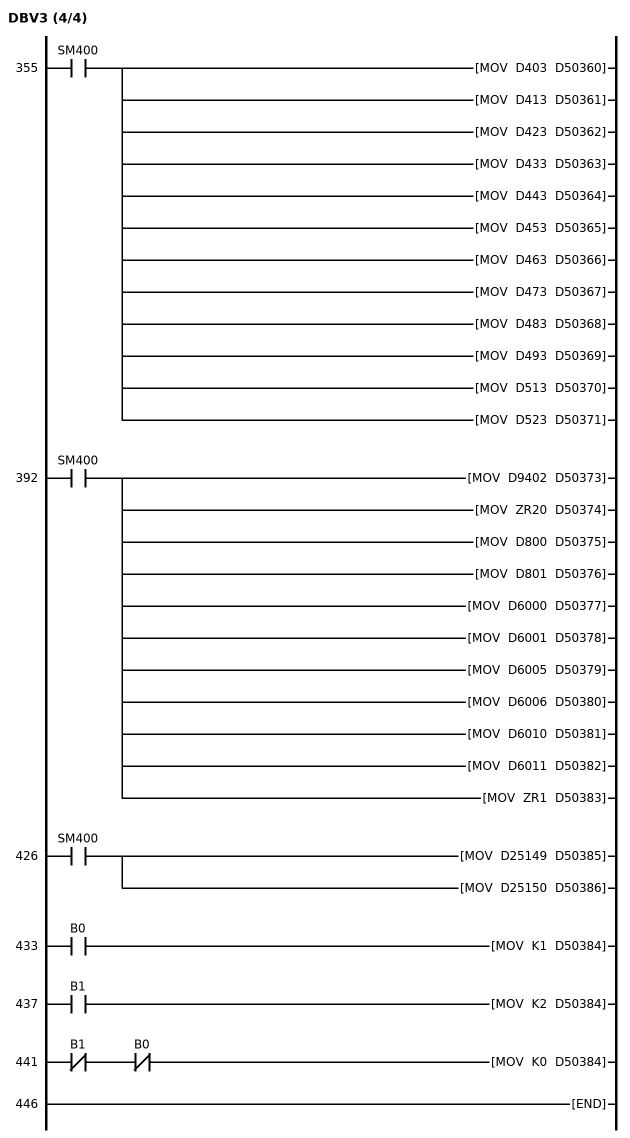
[picture p168: ladder of DBV3, rungs at steps 355 to 446]
355   LD      SM400
      MOV     D403 D50360
      MOV     D413 D50361
      MOV     D423 D50362
      MOV     D433 D50363
      MOV     D443 D50364
      MOV     D453 D50365
      MOV     D463 D50366
      MOV     D473 D50367
      MOV     D483 D50368
      MOV     D493 D50369
      MOV     D513 D50370
      MOV     D523 D50371
392   LD      SM400
      MOV     D9402 D50373
      MOV     ZR20 D50374
      MOV     D800 D50375
      MOV     D801 D50376
      MOV     D6000 D50377
      MOV     D6001 D50378
      MOV     D6005 D50379
      MOV     D6006 D50380
      MOV     D6010 D50381
      MOV     D6011 D50382
      MOV     ZR1 D50383
426   LD      SM400
      MOV     D25149 D50385
      MOV     D25150 D50386
433   LD      B0
      MOV     K1 D50384
437   LD      B1
      MOV     K2 D50384
441   LDI     B1
      ANI     B0
      MOV     K0 D50384
446   END
END_PROGRAM

PROGRAM dryer_cover
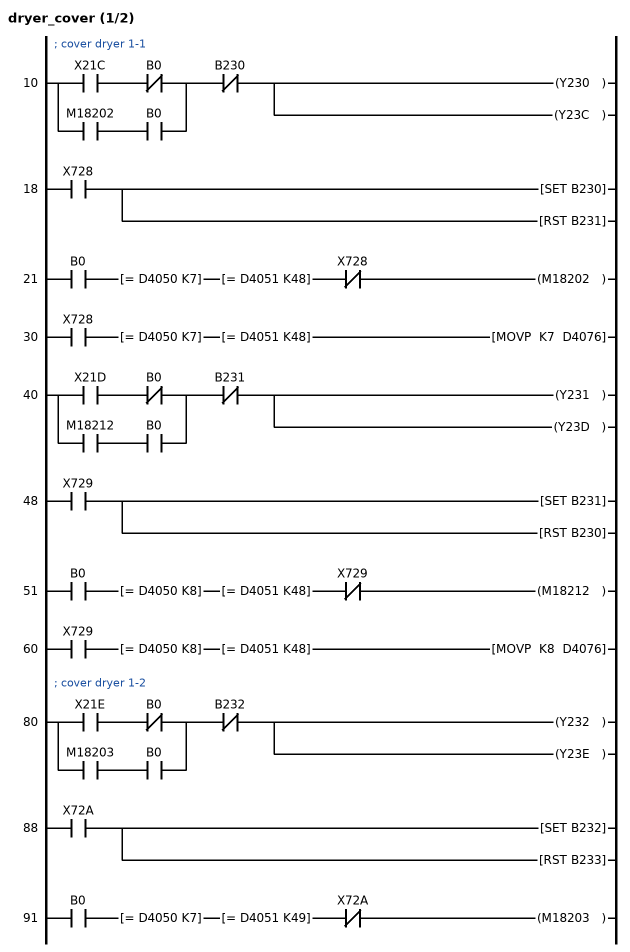
; cover dryer 1-1
10    LD      X21C
      ANI     B0
      LD      M18202
      AND     B0
      ORB
      ANI     B230
      OUT     Y230
      OUT     Y23C
18    LD      X728
      SET     B230
      RST     B231
21    LD      B0
      AND=    D4050 K7
      AND=    D4051 K48
      ANI     X728
      OUT     M18202
30    LD      X728
      AND=    D4050 K7
      AND=    D4051 K48
      MOVP    K7 D4076
40    LD      X21D
      ANI     B0
      LD      M18212
      AND     B0
      ORB
      ANI     B231
      OUT     Y231
      OUT     Y23D
48    LD      X729
      SET     B231
      RST     B230
51    LD      B0
      AND=    D4050 K8
      AND=    D4051 K48
      ANI     X729
      OUT     M18212
60    LD      X729
      AND=    D4050 K8
      AND=    D4051 K48
      MOVP    K8 D4076
; cover dryer 1-2
80    LD      X21E
      ANI     B0
      LD      M18203
      AND     B0
      ORB
      ANI     B232
      OUT     Y232
      OUT     Y23E
88    LD      X72A
      SET     B232
      RST     B233
91    LD      B0
      AND=    D4050 K7
      AND=    D4051 K49
      ANI     X72A
      OUT     M18203
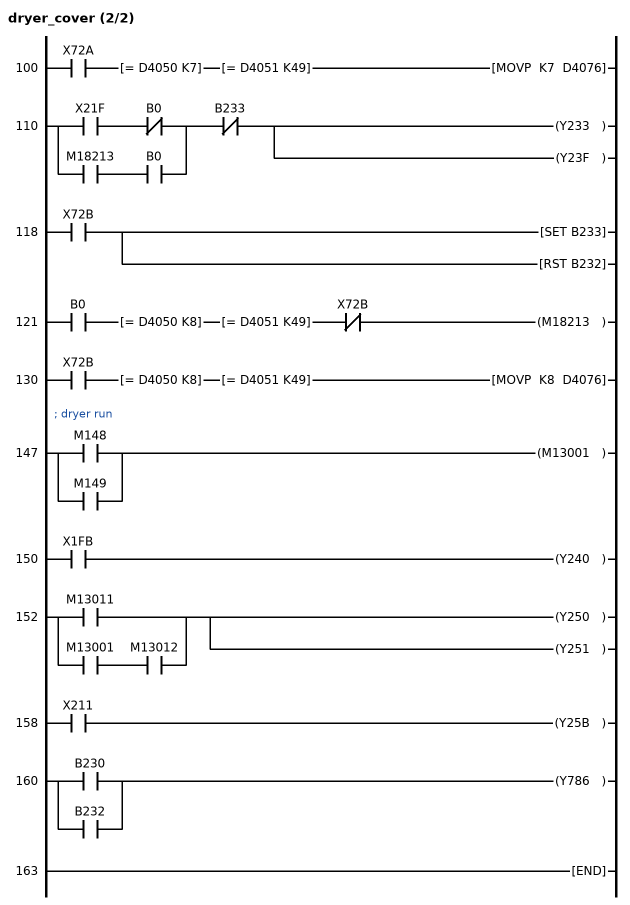
100   LD      X72A
      AND=    D4050 K7
      AND=    D4051 K49
      MOVP    K7 D4076
110   LD      X21F
      ANI     B0
      LD      M18213
      AND     B0
      ORB
      ANI     B233
      OUT     Y233
      OUT     Y23F
118   LD      X72B
      SET     B233
      RST     B232
121   LD      B0
      AND=    D4050 K8
      AND=    D4051 K49
      ANI     X72B
      OUT     M18213
130   LD      X72B
      AND=    D4050 K8
      AND=    D4051 K49
      MOVP    K8 D4076
; dryer run
147   LD      M148
      OR      M149
      OUT     M13001
150   LD      X1FB
      OUT     Y240
152   LD      M13011
      LD      M13001
      AND     M13012
      ORB
      OUT     Y250
      OUT     Y251
158   LD      X211
      OUT     Y25B
160   LD      B230
      OR      B232
      OUT     Y786
163   END
END_PROGRAM

FUNCTION_BLOCK I+ST_4f96081e274e4d1c
VAR_INPUT
  __IST_EN_IN : BOOL;
END_VAR
VAR_OUTPUT
  __IST_EN_OUT : BOOL;
END_VAR
(* IST HEADER START *)
IF NOT __IST_EN_IN THEN __IST_EN_OUT:=FALSE; RETURN; END_IF;
(* VERSION=1:TYPE=STB *)
(* IST HEADER END *)
D3016 := D3006 / k10 ;
END_FUNCTION_BLOCK

FUNCTION_BLOCK I+ST_76367eaf8b844e8d
VAR_INPUT
  __IST_EN_IN : BOOL;
END_VAR
VAR_OUTPUT
  __IST_EN_OUT : BOOL;
END_VAR
(* IST HEADER START *)
IF NOT __IST_EN_IN THEN __IST_EN_OUT:=FALSE; RETURN; END_IF;
(* VERSION=1:TYPE=STB *)
(* IST HEADER END *)
D3015 := D3006 / k10 ;
END_FUNCTION_BLOCK

FUNCTION_BLOCK I+ST_b7c0c6d72a974ae8
VAR_INPUT
  __IST_EN_IN : BOOL;
END_VAR
VAR_OUTPUT
  __IST_EN_OUT : BOOL;
END_VAR
(* IST HEADER START *)
IF NOT __IST_EN_IN THEN __IST_EN_OUT:=FALSE; RETURN; END_IF;
(* VERSION=1:TYPE=STB *)
(* IST HEADER END *)
ZR1010000Z9 := k0 ;
ZR1020000Z9:= k0 ;
ZR1030000Z9 := k0 ;
ZR1040000Z9 := k0 ;
ZR1050000Z9 := k0 ;
ZR1060000Z9 := k0 ;
ZR1070000Z9 := k0 ;
ZR1080000Z9 := k0 ;
ZR1090000Z9 := k0 ;
ZR1100000Z9 := k0 ;
ZR1110000Z9 := k0 ;
ZR1120000Z9 := k0 ;
ZR1130000Z9 := k0 ;
ZR1140000Z9 := k0 ;
ZR1150000Z9 := k0 ;
ZR1160000Z9 := k0 ;
ZR1170000Z9 := k0 ;
ZR1180000Z9 := k0 ;
ZR1190000Z9 := k0 ;
ZR1200000Z9 := k0 ;
ZR1210000Z9 := k0 ;
ZR1220000Z9 := k0 ;
ZR1230000Z9 := k0 ;
ZR1240000Z9 := k0 ;
ZR1250000Z9 := k0 ;
ZR1260000Z9 := k0 ;
ZR1270000Z9 := k0 ;
ZR1280000Z9 := k0 ;
ZR1290000Z9 := k0 ;
ZR1300000Z9 := k0 ;
ZR1310000Z9 := k0 ;
ZR1320000Z9 := k0 ;
ZR1330000Z9 := k0 ;
ZR1340000Z9 := k0 ;
ZR1350000Z9 := k0 ;
ZR1360000Z9 := k0 ;
ZR1370000Z9 := k0 ;
ZR1380000Z9 := k0 ;
ZR1390000Z9 := k0 ;
ZR1400000Z9 := k0 ;
ZR1410000Z9 := k0 ;
ZR1420000Z9 := k0 ;
ZR1430000Z9 := k0 ;
ZR1440000Z9 := k0 ;
ZR1450000Z9 := k0 ;
ZR1460000Z9 := k0 ;
ZR1470000Z9 := k0 ;
ZR1480000Z9 := k0 ;
ZR1490000Z9 := k0 ;
ZR1500000Z9 := k0 ;
ZR1510000Z9 := k0 ;
ZR1520000Z9 := k0 ;
ZR1530000Z9 := k0 ;
ZR1540000Z9 := k0 ;
ZR1550000Z9 := k0 ;
ZR1560000Z9 := k0 ;
ZR1570000Z9 := k0 ;
ZR1580000Z9 := k0 ;
ZR1590000Z9 := k0 ;
ZR1600000Z9 := k0 ;
END_FUNCTION_BLOCK

FUNCTION_BLOCK I+ST_f649ea45d16546a8
VAR_INPUT
  __IST_EN_IN : BOOL;
END_VAR
VAR_OUTPUT
  __IST_EN_OUT : BOOL;
END_VAR
(* IST HEADER START *)
IF NOT __IST_EN_IN THEN __IST_EN_OUT:=FALSE; RETURN; END_IF;
(* VERSION=1:TYPE=STB *)
(* IST HEADER END *)
ZR1610000Z9 := k0 ;
ZR1620000Z9 := k0 ;
ZR1630000Z9 := k0 ;
ZR1640000Z9 := k0 ;
ZR1650000Z9 := k0 ;
ZR1660000Z9 := k0 ;
ZR1670000Z9 := k0 ;
ZR1680000Z9 := k0 ;
ZR1690000Z9 := k0 ;

ZR1800000Z9 := k0 ;
ZR1810000Z9 := k0 ;
ZR1820000Z9 := k0 ;
ZR1830000Z9 := k0 ;
ZR1840000Z9 := k0 ;
ZR1850000Z9 := k0 ;
ZR1860000Z9 := k0 ;
ZR1870000Z9 := k0 ;
ZR1880000Z9 := k0 ;
ZR1890000Z9 := k0 ;
ZR1900000Z9 := k0 ;
END_FUNCTION_BLOCK

PROGRAM POU_01
0     END
END_PROGRAM

PROGRAM pro_time
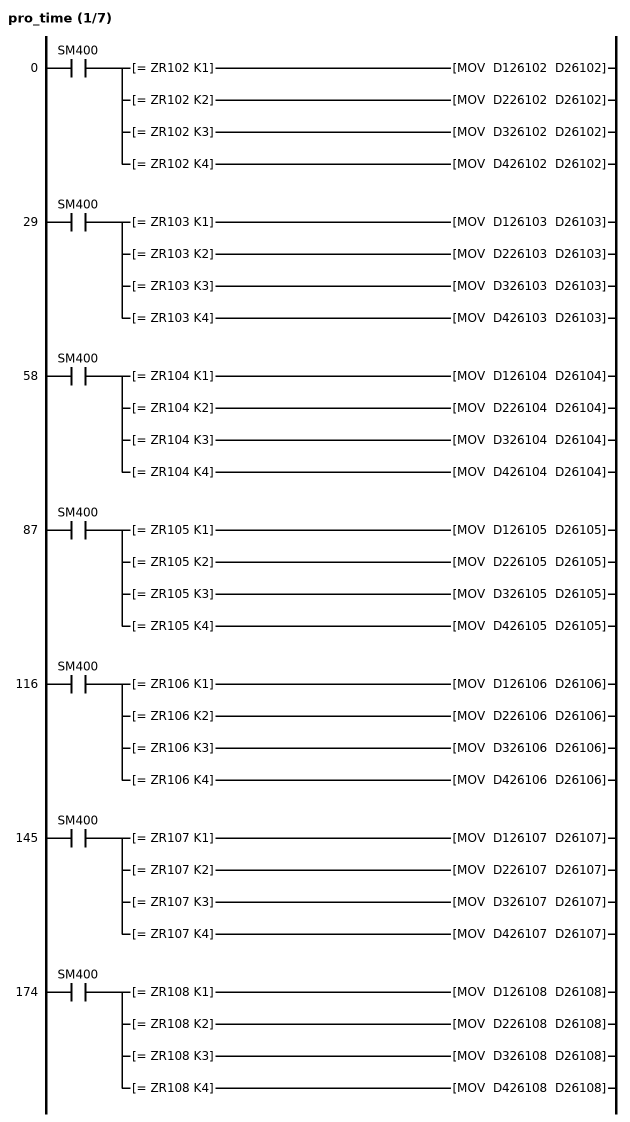
0     LD      SM400
      MPS
      AND=    ZR102 K1
      MOV     D126102 D26102
      MRD
      AND=    ZR102 K2
      MOV     D226102 D26102
      MRD
      AND=    ZR102 K3
      MOV     D326102 D26102
      MPP
      AND=    ZR102 K4
      MOV     D426102 D26102
29    LD      SM400
      MPS
      AND=    ZR103 K1
      MOV     D126103 D26103
      MRD
      AND=    ZR103 K2
      MOV     D226103 D26103
      MRD
      AND=    ZR103 K3
      MOV     D326103 D26103
      MPP
      AND=    ZR103 K4
      MOV     D426103 D26103
58    LD      SM400
      MPS
      AND=    ZR104 K1
      MOV     D126104 D26104
      MRD
      AND=    ZR104 K2
      MOV     D226104 D26104
      MRD
      AND=    ZR104 K3
      MOV     D326104 D26104
      MPP
      AND=    ZR104 K4
      MOV     D426104 D26104
87    LD      SM400
      MPS
      AND=    ZR105 K1
      MOV     D126105 D26105
      MRD
      AND=    ZR105 K2
      MOV     D226105 D26105
      MRD
      AND=    ZR105 K3
      MOV     D326105 D26105
      MPP
      AND=    ZR105 K4
      MOV     D426105 D26105
116   LD      SM400
      MPS
      AND=    ZR106 K1
      MOV     D126106 D26106
      MRD
      AND=    ZR106 K2
      MOV     D226106 D26106
      MRD
      AND=    ZR106 K3
      MOV     D326106 D26106
      MPP
      AND=    ZR106 K4
      MOV     D426106 D26106
145   LD      SM400
      MPS
      AND=    ZR107 K1
      MOV     D126107 D26107
      MRD
      AND=    ZR107 K2
      MOV     D226107 D26107
      MRD
      AND=    ZR107 K3
      MOV     D326107 D26107
      MPP
      AND=    ZR107 K4
      MOV     D426107 D26107
174   LD      SM400
      MPS
      AND=    ZR108 K1
      MOV     D126108 D26108
      MRD
      AND=    ZR108 K2
      MOV     D226108 D26108
      MRD
      AND=    ZR108 K3
      MOV     D326108 D26108
      MPP
      AND=    ZR108 K4
      MOV     D426108 D26108
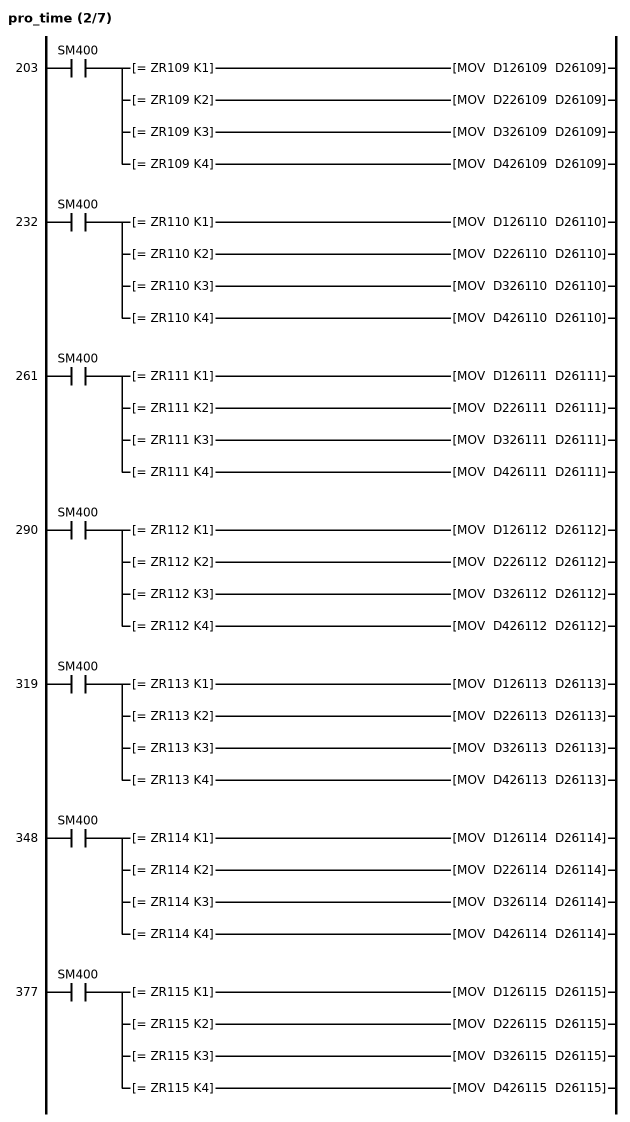
203   LD      SM400
      MPS
      AND=    ZR109 K1
      MOV     D126109 D26109
      MRD
      AND=    ZR109 K2
      MOV     D226109 D26109
      MRD
      AND=    ZR109 K3
      MOV     D326109 D26109
      MPP
      AND=    ZR109 K4
      MOV     D426109 D26109
232   LD      SM400
      MPS
      AND=    ZR110 K1
      MOV     D126110 D26110
      MRD
      AND=    ZR110 K2
      MOV     D226110 D26110
      MRD
      AND=    ZR110 K3
      MOV     D326110 D26110
      MPP
      AND=    ZR110 K4
      MOV     D426110 D26110
261   LD      SM400
      MPS
      AND=    ZR111 K1
      MOV     D126111 D26111
      MRD
      AND=    ZR111 K2
      MOV     D226111 D26111
      MRD
      AND=    ZR111 K3
      MOV     D326111 D26111
      MPP
      AND=    ZR111 K4
      MOV     D426111 D26111
290   LD      SM400
      MPS
      AND=    ZR112 K1
      MOV     D126112 D26112
      MRD
      AND=    ZR112 K2
      MOV     D226112 D26112
      MRD
      AND=    ZR112 K3
      MOV     D326112 D26112
      MPP
      AND=    ZR112 K4
      MOV     D426112 D26112
319   LD      SM400
      MPS
      AND=    ZR113 K1
      MOV     D126113 D26113
      MRD
      AND=    ZR113 K2
      MOV     D226113 D26113
      MRD
      AND=    ZR113 K3
      MOV     D326113 D26113
      MPP
      AND=    ZR113 K4
      MOV     D426113 D26113
348   LD      SM400
      MPS
      AND=    ZR114 K1
      MOV     D126114 D26114
      MRD
      AND=    ZR114 K2
      MOV     D226114 D26114
      MRD
      AND=    ZR114 K3
      MOV     D326114 D26114
      MPP
      AND=    ZR114 K4
      MOV     D426114 D26114
377   LD      SM400
      MPS
      AND=    ZR115 K1
      MOV     D126115 D26115
      MRD
      AND=    ZR115 K2
      MOV     D226115 D26115
      MRD
      AND=    ZR115 K3
      MOV     D326115 D26115
      MPP
      AND=    ZR115 K4
      MOV     D426115 D26115
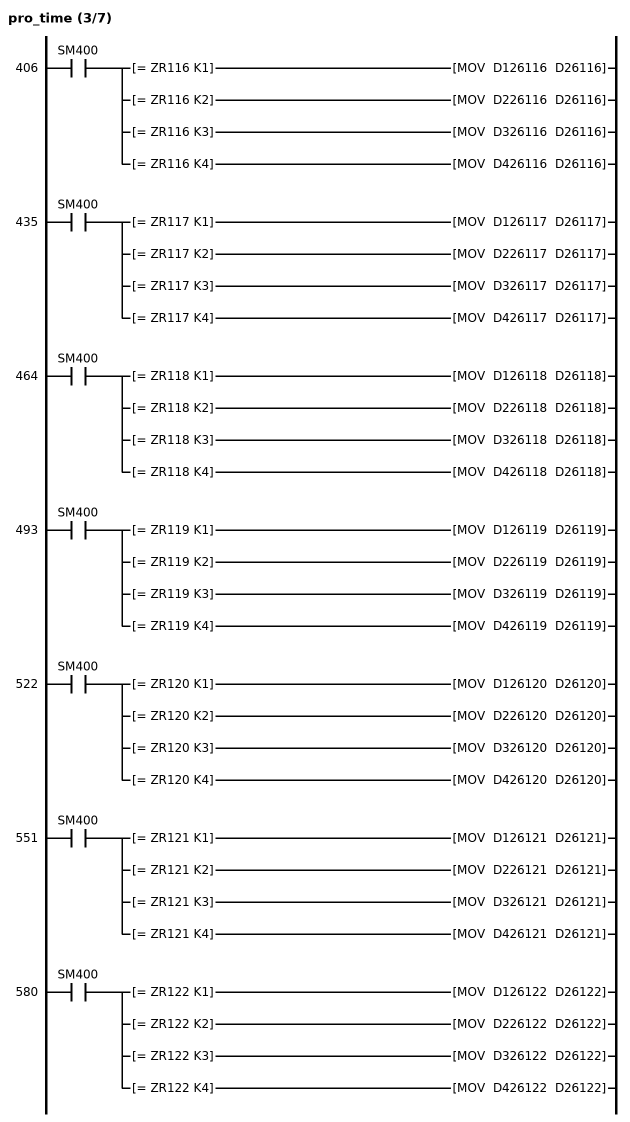
406   LD      SM400
      MPS
      AND=    ZR116 K1
      MOV     D126116 D26116
      MRD
      AND=    ZR116 K2
      MOV     D226116 D26116
      MRD
      AND=    ZR116 K3
      MOV     D326116 D26116
      MPP
      AND=    ZR116 K4
      MOV     D426116 D26116
435   LD      SM400
      MPS
      AND=    ZR117 K1
      MOV     D126117 D26117
      MRD
      AND=    ZR117 K2
      MOV     D226117 D26117
      MRD
      AND=    ZR117 K3
      MOV     D326117 D26117
      MPP
      AND=    ZR117 K4
      MOV     D426117 D26117
464   LD      SM400
      MPS
      AND=    ZR118 K1
      MOV     D126118 D26118
      MRD
      AND=    ZR118 K2
      MOV     D226118 D26118
      MRD
      AND=    ZR118 K3
      MOV     D326118 D26118
      MPP
      AND=    ZR118 K4
      MOV     D426118 D26118
493   LD      SM400
      MPS
      AND=    ZR119 K1
      MOV     D126119 D26119
      MRD
      AND=    ZR119 K2
      MOV     D226119 D26119
      MRD
      AND=    ZR119 K3
      MOV     D326119 D26119
      MPP
      AND=    ZR119 K4
      MOV     D426119 D26119
522   LD      SM400
      MPS
      AND=    ZR120 K1
      MOV     D126120 D26120
      MRD
      AND=    ZR120 K2
      MOV     D226120 D26120
      MRD
      AND=    ZR120 K3
      MOV     D326120 D26120
      MPP
      AND=    ZR120 K4
      MOV     D426120 D26120
551   LD      SM400
      MPS
      AND=    ZR121 K1
      MOV     D126121 D26121
      MRD
      AND=    ZR121 K2
      MOV     D226121 D26121
      MRD
      AND=    ZR121 K3
      MOV     D326121 D26121
      MPP
      AND=    ZR121 K4
      MOV     D426121 D26121
580   LD      SM400
      MPS
      AND=    ZR122 K1
      MOV     D126122 D26122
      MRD
      AND=    ZR122 K2
      MOV     D226122 D26122
      MRD
      AND=    ZR122 K3
      MOV     D326122 D26122
      MPP
      AND=    ZR122 K4
      MOV     D426122 D26122
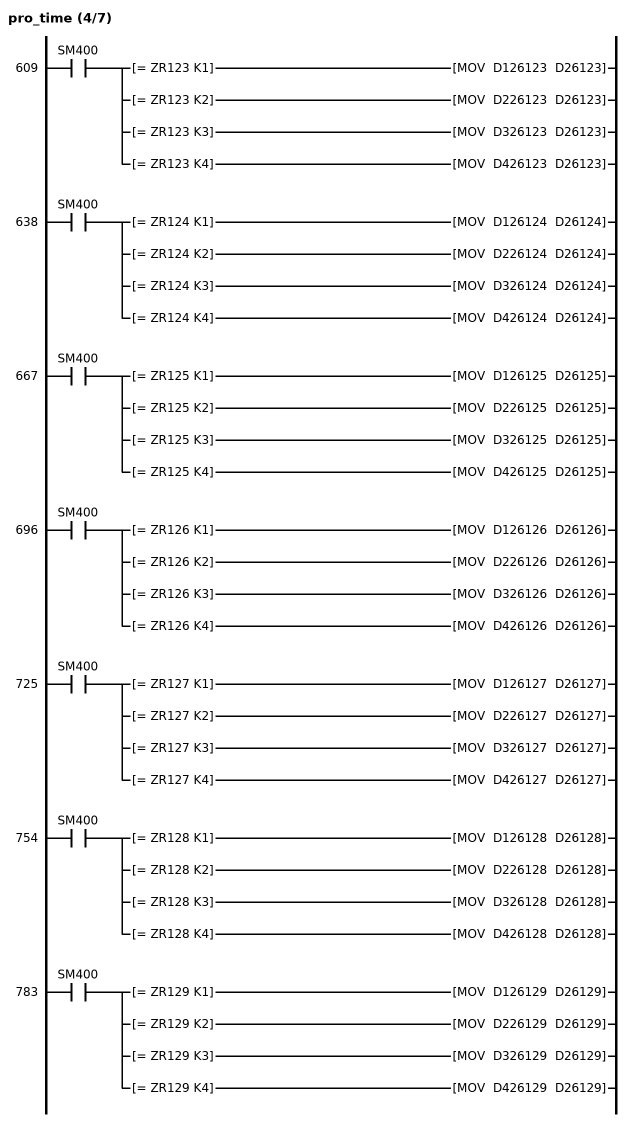
609   LD      SM400
      MPS
      AND=    ZR123 K1
      MOV     D126123 D26123
      MRD
      AND=    ZR123 K2
      MOV     D226123 D26123
      MRD
      AND=    ZR123 K3
      MOV     D326123 D26123
      MPP
      AND=    ZR123 K4
      MOV     D426123 D26123
638   LD      SM400
      MPS
      AND=    ZR124 K1
      MOV     D126124 D26124
      MRD
      AND=    ZR124 K2
      MOV     D226124 D26124
      MRD
      AND=    ZR124 K3
      MOV     D326124 D26124
      MPP
      AND=    ZR124 K4
      MOV     D426124 D26124
667   LD      SM400
      MPS
      AND=    ZR125 K1
      MOV     D126125 D26125
      MRD
      AND=    ZR125 K2
      MOV     D226125 D26125
      MRD
      AND=    ZR125 K3
      MOV     D326125 D26125
      MPP
      AND=    ZR125 K4
      MOV     D426125 D26125
696   LD      SM400
      MPS
      AND=    ZR126 K1
      MOV     D126126 D26126
      MRD
      AND=    ZR126 K2
      MOV     D226126 D26126
      MRD
      AND=    ZR126 K3
      MOV     D326126 D26126
      MPP
      AND=    ZR126 K4
      MOV     D426126 D26126
725   LD      SM400
      MPS
      AND=    ZR127 K1
      MOV     D126127 D26127
      MRD
      AND=    ZR127 K2
      MOV     D226127 D26127
      MRD
      AND=    ZR127 K3
      MOV     D326127 D26127
      MPP
      AND=    ZR127 K4
      MOV     D426127 D26127
754   LD      SM400
      MPS
      AND=    ZR128 K1
      MOV     D126128 D26128
      MRD
      AND=    ZR128 K2
      MOV     D226128 D26128
      MRD
      AND=    ZR128 K3
      MOV     D326128 D26128
      MPP
      AND=    ZR128 K4
      MOV     D426128 D26128
783   LD      SM400
      MPS
      AND=    ZR129 K1
      MOV     D126129 D26129
      MRD
      AND=    ZR129 K2
      MOV     D226129 D26129
      MRD
      AND=    ZR129 K3
      MOV     D326129 D26129
      MPP
      AND=    ZR129 K4
      MOV     D426129 D26129
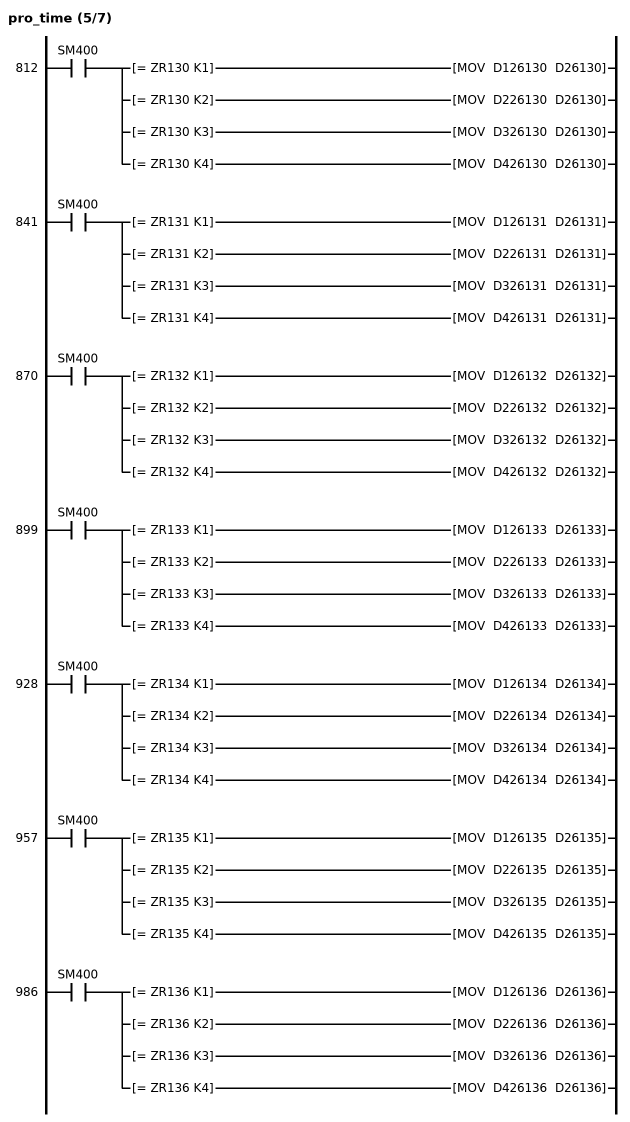
812   LD      SM400
      MPS
      AND=    ZR130 K1
      MOV     D126130 D26130
      MRD
      AND=    ZR130 K2
      MOV     D226130 D26130
      MRD
      AND=    ZR130 K3
      MOV     D326130 D26130
      MPP
      AND=    ZR130 K4
      MOV     D426130 D26130
841   LD      SM400
      MPS
      AND=    ZR131 K1
      MOV     D126131 D26131
      MRD
      AND=    ZR131 K2
      MOV     D226131 D26131
      MRD
      AND=    ZR131 K3
      MOV     D326131 D26131
      MPP
      AND=    ZR131 K4
      MOV     D426131 D26131
870   LD      SM400
      MPS
      AND=    ZR132 K1
      MOV     D126132 D26132
      MRD
      AND=    ZR132 K2
      MOV     D226132 D26132
      MRD
      AND=    ZR132 K3
      MOV     D326132 D26132
      MPP
      AND=    ZR132 K4
      MOV     D426132 D26132
899   LD      SM400
      MPS
      AND=    ZR133 K1
      MOV     D126133 D26133
      MRD
      AND=    ZR133 K2
      MOV     D226133 D26133
      MRD
      AND=    ZR133 K3
      MOV     D326133 D26133
      MPP
      AND=    ZR133 K4
      MOV     D426133 D26133
928   LD      SM400
      MPS
      AND=    ZR134 K1
      MOV     D126134 D26134
      MRD
      AND=    ZR134 K2
      MOV     D226134 D26134
      MRD
      AND=    ZR134 K3
      MOV     D326134 D26134
      MPP
      AND=    ZR134 K4
      MOV     D426134 D26134
957   LD      SM400
      MPS
      AND=    ZR135 K1
      MOV     D126135 D26135
      MRD
      AND=    ZR135 K2
      MOV     D226135 D26135
      MRD
      AND=    ZR135 K3
      MOV     D326135 D26135
      MPP
      AND=    ZR135 K4
      MOV     D426135 D26135
986   LD      SM400
      MPS
      AND=    ZR136 K1
      MOV     D126136 D26136
      MRD
      AND=    ZR136 K2
      MOV     D226136 D26136
      MRD
      AND=    ZR136 K3
      MOV     D326136 D26136
      MPP
      AND=    ZR136 K4
      MOV     D426136 D26136
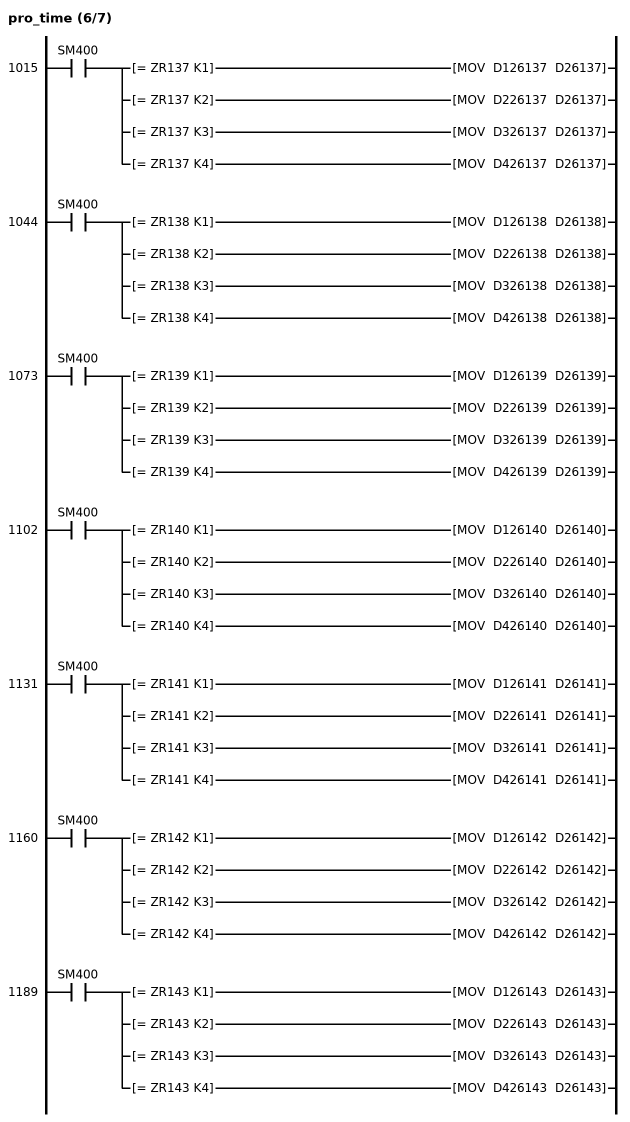
1015  LD      SM400
      MPS
      AND=    ZR137 K1
      MOV     D126137 D26137
      MRD
      AND=    ZR137 K2
      MOV     D226137 D26137
      MRD
      AND=    ZR137 K3
      MOV     D326137 D26137
      MPP
      AND=    ZR137 K4
      MOV     D426137 D26137
1044  LD      SM400
      MPS
      AND=    ZR138 K1
      MOV     D126138 D26138
      MRD
      AND=    ZR138 K2
      MOV     D226138 D26138
      MRD
      AND=    ZR138 K3
      MOV     D326138 D26138
      MPP
      AND=    ZR138 K4
      MOV     D426138 D26138
1073  LD      SM400
      MPS
      AND=    ZR139 K1
      MOV     D126139 D26139
      MRD
      AND=    ZR139 K2
      MOV     D226139 D26139
      MRD
      AND=    ZR139 K3
      MOV     D326139 D26139
      MPP
      AND=    ZR139 K4
      MOV     D426139 D26139
1102  LD      SM400
      MPS
      AND=    ZR140 K1
      MOV     D126140 D26140
      MRD
      AND=    ZR140 K2
      MOV     D226140 D26140
      MRD
      AND=    ZR140 K3
      MOV     D326140 D26140
      MPP
      AND=    ZR140 K4
      MOV     D426140 D26140
1131  LD      SM400
      MPS
      AND=    ZR141 K1
      MOV     D126141 D26141
      MRD
      AND=    ZR141 K2
      MOV     D226141 D26141
      MRD
      AND=    ZR141 K3
      MOV     D326141 D26141
      MPP
      AND=    ZR141 K4
      MOV     D426141 D26141
1160  LD      SM400
      MPS
      AND=    ZR142 K1
      MOV     D126142 D26142
      MRD
      AND=    ZR142 K2
      MOV     D226142 D26142
      MRD
      AND=    ZR142 K3
      MOV     D326142 D26142
      MPP
      AND=    ZR142 K4
      MOV     D426142 D26142
1189  LD      SM400
      MPS
      AND=    ZR143 K1
      MOV     D126143 D26143
      MRD
      AND=    ZR143 K2
      MOV     D226143 D26143
      MRD
      AND=    ZR143 K3
      MOV     D326143 D26143
      MPP
      AND=    ZR143 K4
      MOV     D426143 D26143
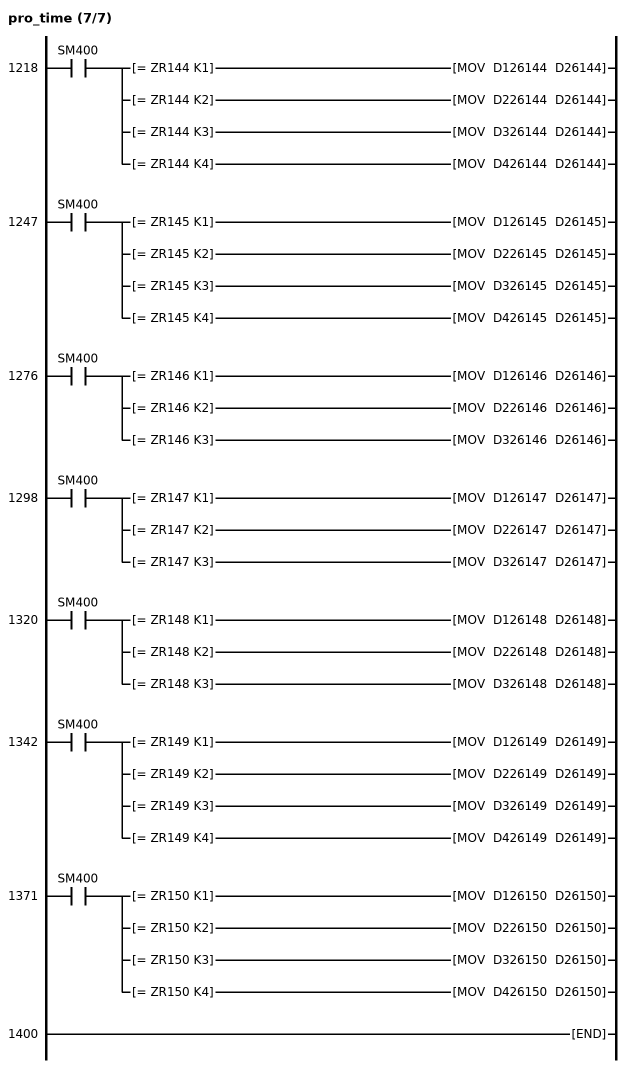
1218  LD      SM400
      MPS
      AND=    ZR144 K1
      MOV     D126144 D26144
      MRD
      AND=    ZR144 K2
      MOV     D226144 D26144
      MRD
      AND=    ZR144 K3
      MOV     D326144 D26144
      MPP
      AND=    ZR144 K4
      MOV     D426144 D26144
1247  LD      SM400
      MPS
      AND=    ZR145 K1
      MOV     D126145 D26145
      MRD
      AND=    ZR145 K2
      MOV     D226145 D26145
      MRD
      AND=    ZR145 K3
      MOV     D326145 D26145
      MPP
      AND=    ZR145 K4
      MOV     D426145 D26145
1276  LD      SM400
      MPS
      AND=    ZR146 K1
      MOV     D126146 D26146
      MRD
      AND=    ZR146 K2
      MOV     D226146 D26146
      MPP
      AND=    ZR146 K3
      MOV     D326146 D26146
1298  LD      SM400
      MPS
      AND=    ZR147 K1
      MOV     D126147 D26147
      MRD
      AND=    ZR147 K2
      MOV     D226147 D26147
      MPP
      AND=    ZR147 K3
      MOV     D326147 D26147
1320  LD      SM400
      MPS
      AND=    ZR148 K1
      MOV     D126148 D26148
      MRD
      AND=    ZR148 K2
      MOV     D226148 D26148
      MPP
      AND=    ZR148 K3
      MOV     D326148 D26148
1342  LD      SM400
      MPS
      AND=    ZR149 K1
      MOV     D126149 D26149
      MRD
      AND=    ZR149 K2
      MOV     D226149 D26149
      MRD
      AND=    ZR149 K3
      MOV     D326149 D26149
      MPP
      AND=    ZR149 K4
      MOV     D426149 D26149
1371  LD      SM400
      MPS
      AND=    ZR150 K1
      MOV     D126150 D26150
      MRD
      AND=    ZR150 K2
      MOV     D226150 D26150
      MRD
      AND=    ZR150 K3
      MOV     D326150 D26150
      MPP
      AND=    ZR150 K4
      MOV     D426150 D26150
1400  END
END_PROGRAM

PROGRAM program_calculate
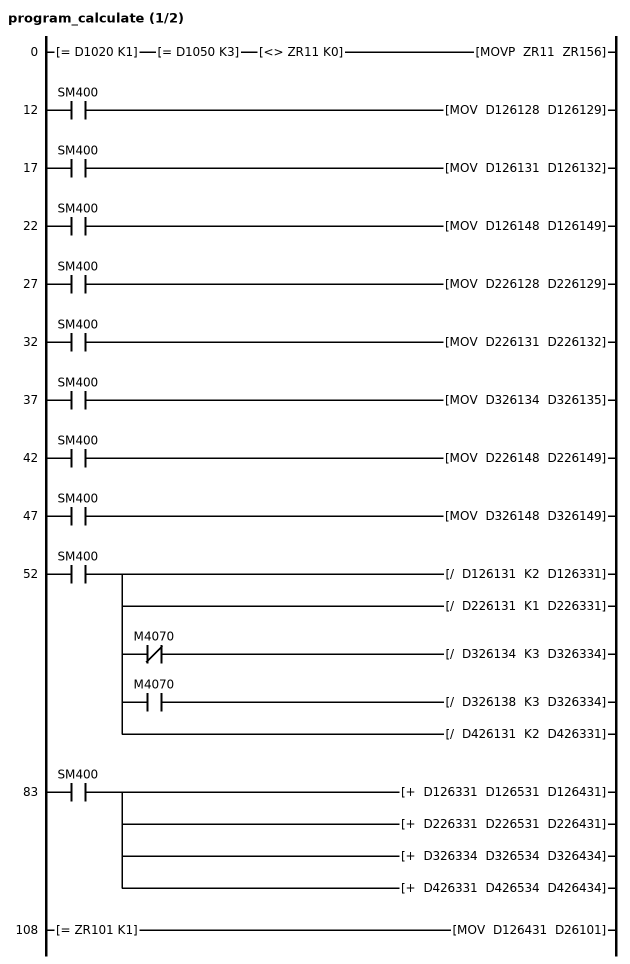
0     LD=     D1020 K1
      AND=    D1050 K3
      AND<>   ZR11 K0
      MOVP    ZR11 ZR156
12    LD      SM400
      MOV     D126128 D126129
17    LD      SM400
      MOV     D126131 D126132
22    LD      SM400
      MOV     D126148 D126149
27    LD      SM400
      MOV     D226128 D226129
32    LD      SM400
      MOV     D226131 D226132
37    LD      SM400
      MOV     D326134 D326135
42    LD      SM400
      MOV     D226148 D226149
47    LD      SM400
      MOV     D326148 D326149
52    LD      SM400
      /       D126131 K2 D126331
      /       D226131 K1 D226331
      MPS
      ANI     M4070
      /       D326134 K3 D326334
      MRD
      AND     M4070
      /       D326138 K3 D326334
      MPP
      /       D426131 K2 D426331
83    LD      SM400
      +       D126331 D126531 D126431
      +       D226331 D226531 D226431
      +       D326334 D326534 D326434
      +       D426331 D426534 D426434
108   LD=     ZR101 K1
      MOV     D126431 D26101
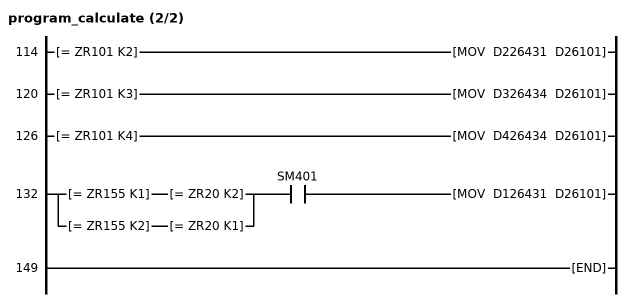
114   LD=     ZR101 K2
      MOV     D226431 D26101
120   LD=     ZR101 K3
      MOV     D326434 D26101
126   LD=     ZR101 K4
      MOV     D426434 D26101
132   LD=     ZR155 K1
      AND=    ZR20 K2
      LD=     ZR155 K2
      AND=    ZR20 K1
      ORB
      AND     SM401
      MOV     D126431 D26101
149   END
END_PROGRAM

PROGRAM pump
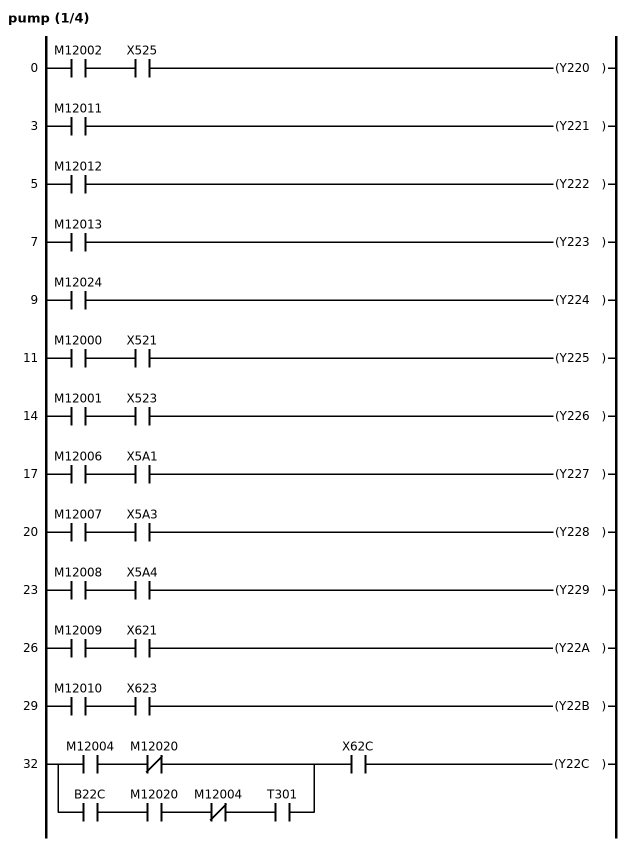
0     LD      M12002
      AND     X525
      OUT     Y220
3     LD      M12011
      OUT     Y221
5     LD      M12012
      OUT     Y222
7     LD      M12013
      OUT     Y223
9     LD      M12024
      OUT     Y224
11    LD      M12000
      AND     X521
      OUT     Y225
14    LD      M12001
      AND     X523
      OUT     Y226
17    LD      M12006
      AND     X5A1
      OUT     Y227
20    LD      M12007
      AND     X5A3
      OUT     Y228
23    LD      M12008
      AND     X5A4
      OUT     Y229
26    LD      M12009
      AND     X621
      OUT     Y22A
29    LD      M12010
      AND     X623
      OUT     Y22B
32    LD      M12004
      ANI     M12020
      LD      B22C
      AND     M12020
      ANI     M12004
      AND     T301
      ORB
      AND     X62C
      OUT     Y22C
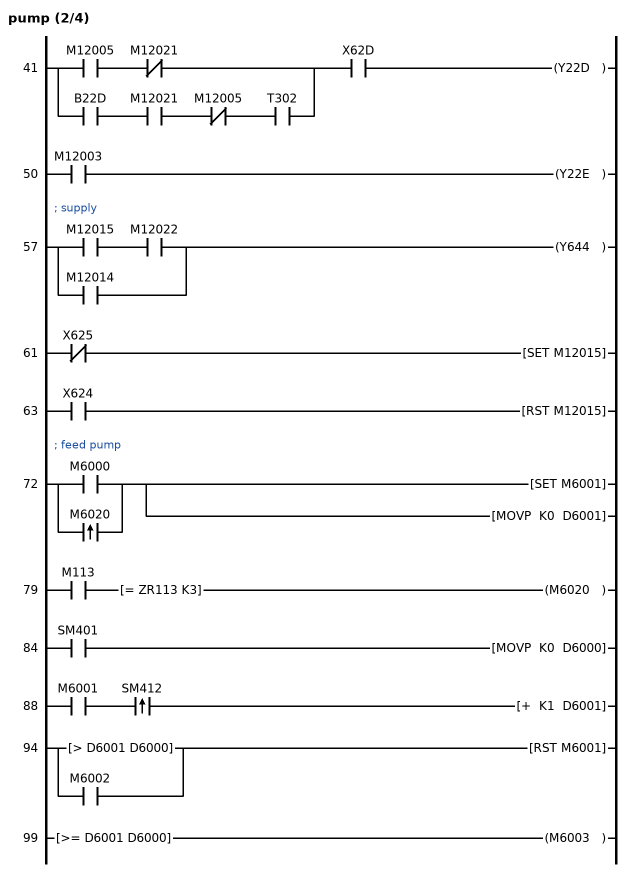
41    LD      M12005
      ANI     M12021
      LD      B22D
      AND     M12021
      ANI     M12005
      AND     T302
      ORB
      AND     X62D
      OUT     Y22D
50    LD      M12003
      OUT     Y22E
; supply
57    LD      M12015
      AND     M12022
      OR      M12014
      OUT     Y644
61    LDI     X625
      SET     M12015
63    LD      X624
      RST     M12015
; feed pump
72    LD      M6000
      ORP     M6020
      SET     M6001
      MOVP    K0 D6001
79    LD      M113
      AND=    ZR113 K3
      OUT     M6020
84    LD      SM401
      MOVP    K0 D6000
88    LD      M6001
      ANDP    SM412
      +       K1 D6001
94    LD>     D6001 D6000
      OR      M6002
      RST     M6001
99    LD>=    D6001 D6000
      OUT     M6003
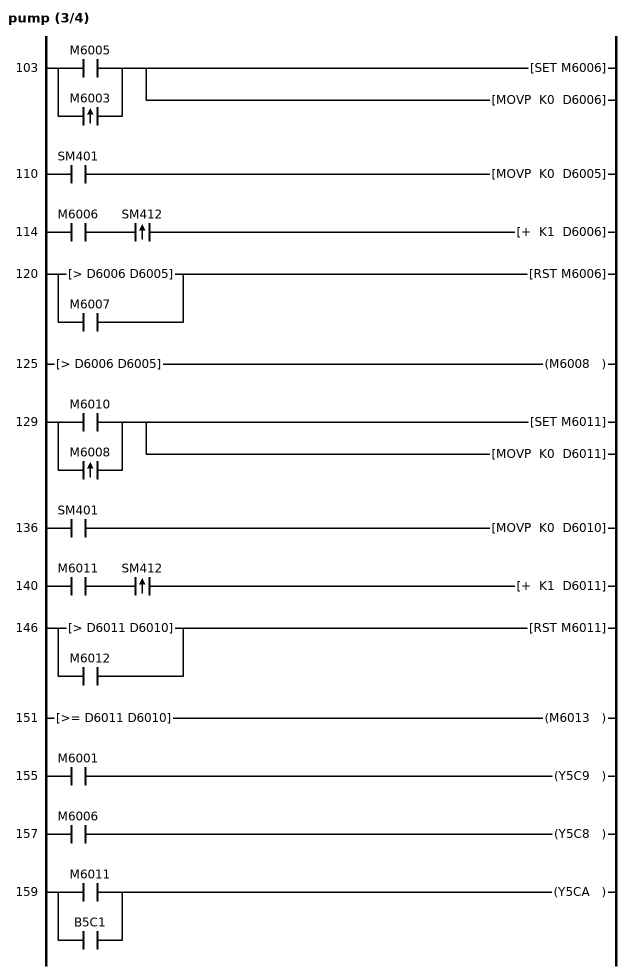
103   LD      M6005
      ORP     M6003
      SET     M6006
      MOVP    K0 D6006
110   LD      SM401
      MOVP    K0 D6005
114   LD      M6006
      ANDP    SM412
      +       K1 D6006
120   LD>     D6006 D6005
      OR      M6007
      RST     M6006
125   LD>     D6006 D6005
      OUT     M6008
129   LD      M6010
      ORP     M6008
      SET     M6011
      MOVP    K0 D6011
136   LD      SM401
      MOVP    K0 D6010
140   LD      M6011
      ANDP    SM412
      +       K1 D6011
146   LD>     D6011 D6010
      OR      M6012
      RST     M6011
151   LD>=    D6011 D6010
      OUT     M6013
155   LD      M6001
      OUT     Y5C9
157   LD      M6006
      OUT     Y5C8
159   LD      M6011
      OR      B5C1
      OUT     Y5CA
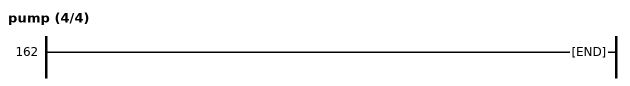
162   END
END_PROGRAM

PROGRAM QC_pass
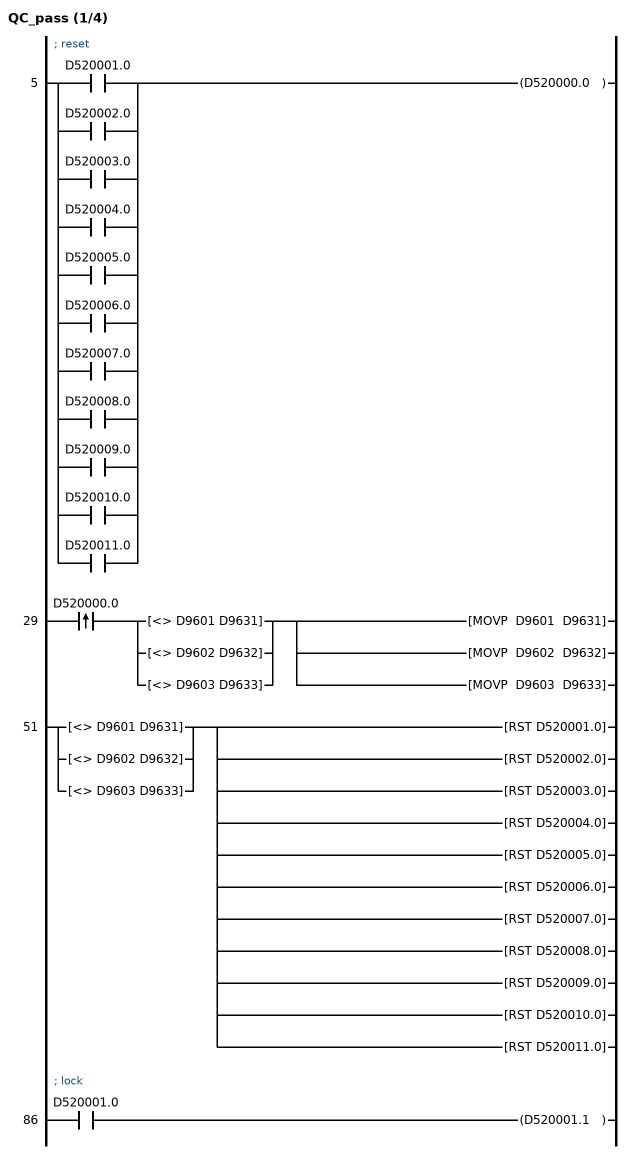
; reset
5     LD      D520001.0
      OR      D520002.0
      OR      D520003.0
      OR      D520004.0
      OR      D520005.0
      OR      D520006.0
      OR      D520007.0
      OR      D520008.0
      OR      D520009.0
      OR      D520010.0
      OR      D520011.0
      OUT     D520000.0
29    LDP     D520000.0
      LD<>    D9601 D9631
      OR<>    D9602 D9632
      OR<>    D9603 D9633
      ANB
      MOVP    D9601 D9631
      MOVP    D9602 D9632
      MOVP    D9603 D9633
51    LD<>    D9601 D9631
      OR<>    D9602 D9632
      OR<>    D9603 D9633
      RST     D520001.0
      RST     D520002.0
      RST     D520003.0
      RST     D520004.0
      RST     D520005.0
      RST     D520006.0
      RST     D520007.0
      RST     D520008.0
      RST     D520009.0
      RST     D520010.0
      RST     D520011.0
; lock
86    LD      D520001.0
      OUT     D520001.1
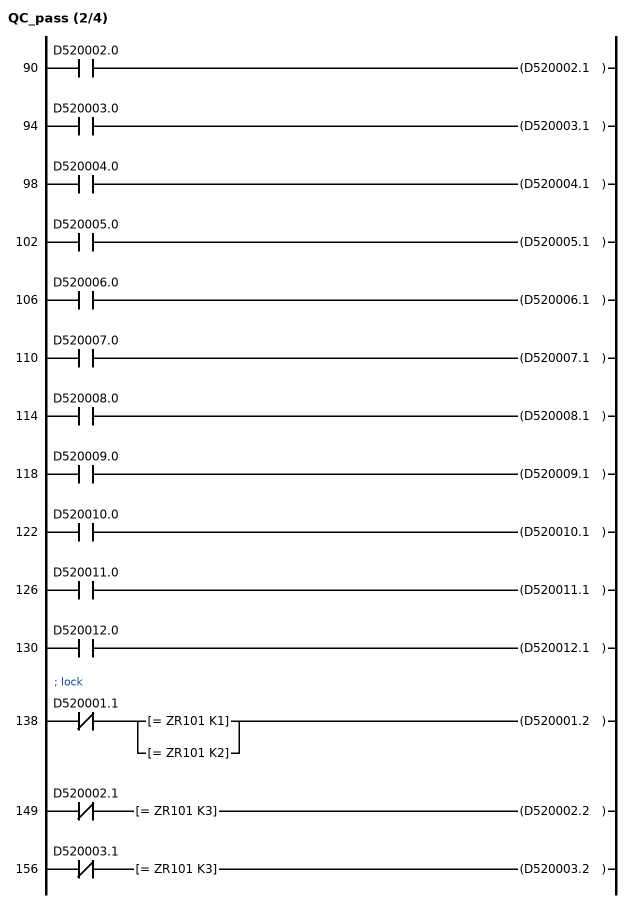
90    LD      D520002.0
      OUT     D520002.1
94    LD      D520003.0
      OUT     D520003.1
98    LD      D520004.0
      OUT     D520004.1
102   LD      D520005.0
      OUT     D520005.1
106   LD      D520006.0
      OUT     D520006.1
110   LD      D520007.0
      OUT     D520007.1
114   LD      D520008.0
      OUT     D520008.1
118   LD      D520009.0
      OUT     D520009.1
122   LD      D520010.0
      OUT     D520010.1
126   LD      D520011.0
      OUT     D520011.1
130   LD      D520012.0
      OUT     D520012.1
; lock
138   LDI     D520001.1
      LD=     ZR101 K1
      OR=     ZR101 K2
      ANB
      OUT     D520001.2
149   LDI     D520002.1
      AND=    ZR101 K3
      OUT     D520002.2
156   LDI     D520003.1
      AND=    ZR101 K3
      OUT     D520003.2
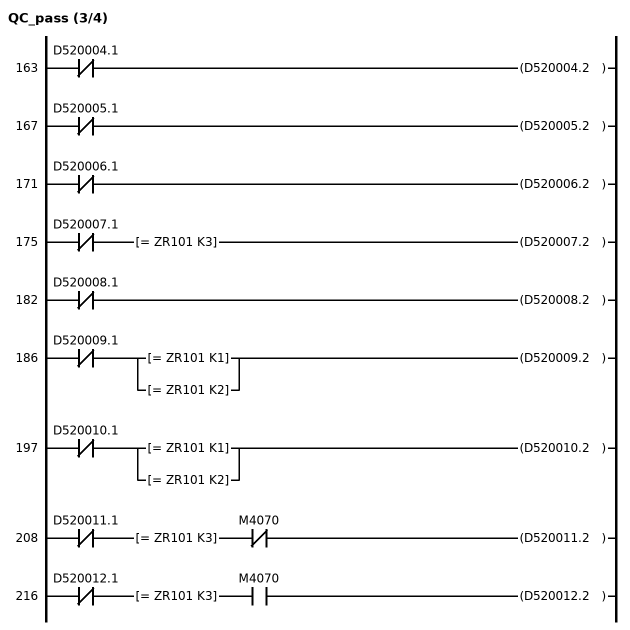
163   LDI     D520004.1
      OUT     D520004.2
167   LDI     D520005.1
      OUT     D520005.2
171   LDI     D520006.1
      OUT     D520006.2
175   LDI     D520007.1
      AND=    ZR101 K3
      OUT     D520007.2
182   LDI     D520008.1
      OUT     D520008.2
186   LDI     D520009.1
      LD=     ZR101 K1
      OR=     ZR101 K2
      ANB
      OUT     D520009.2
197   LDI     D520010.1
      LD=     ZR101 K1
      OR=     ZR101 K2
      ANB
      OUT     D520010.2
208   LDI     D520011.1
      AND=    ZR101 K3
      ANI     M4070
      OUT     D520011.2
216   LDI     D520012.1
      AND=    ZR101 K3
      AND     M4070
      OUT     D520012.2
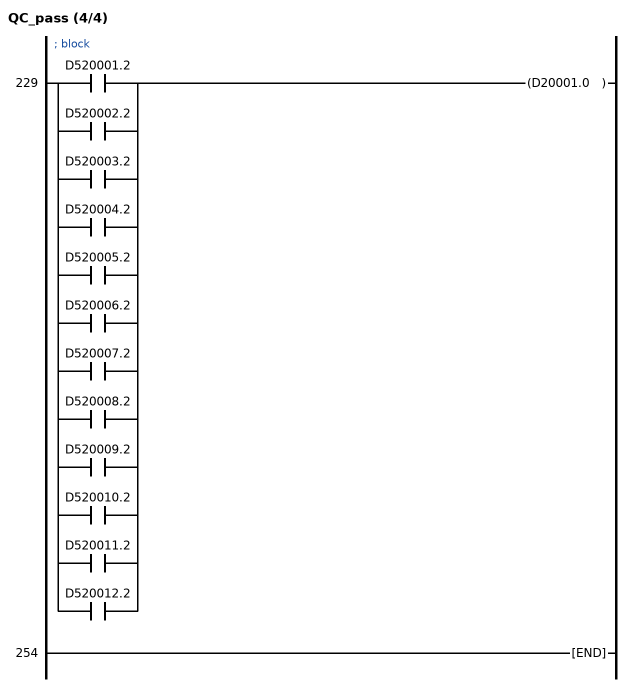
; block
229   LD      D520001.2
      OR      D520002.2
      OR      D520003.2
      OR      D520004.2
      OR      D520005.2
      OR      D520006.2
      OR      D520007.2
      OR      D520008.2
      OR      D520009.2
      OR      D520010.2
      OR      D520011.2
      OR      D520012.2
      OUT     D20001.0
254   END
END_PROGRAM

PROGRAM receive_c
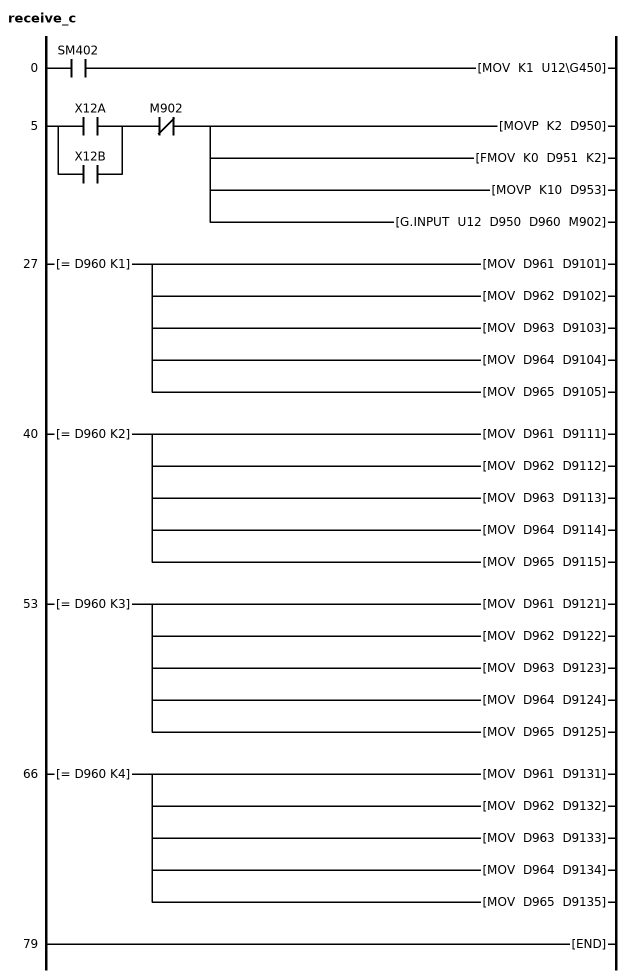
0     LD      SM402
      MOV     K1 U12\G450
5     LD      X12A
      OR      X12B
      ANI     M902
      MOVP    K2 D950
      FMOV    K0 D951 K2
      MOVP    K10 D953
      G.INPUT U12 D950 D960 M902
27    LD=     D960 K1
      MOV     D961 D9101
      MOV     D962 D9102
      MOV     D963 D9103
      MOV     D964 D9104
      MOV     D965 D9105
40    LD=     D960 K2
      MOV     D961 D9111
      MOV     D962 D9112
      MOV     D963 D9113
      MOV     D964 D9114
      MOV     D965 D9115
53    LD=     D960 K3
      MOV     D961 D9121
      MOV     D962 D9122
      MOV     D963 D9123
      MOV     D964 D9124
      MOV     D965 D9125
66    LD=     D960 K4
      MOV     D961 D9131
      MOV     D962 D9132
      MOV     D963 D9133
      MOV     D964 D9134
      MOV     D965 D9135
79    END
END_PROGRAM

PROGRAM rocking
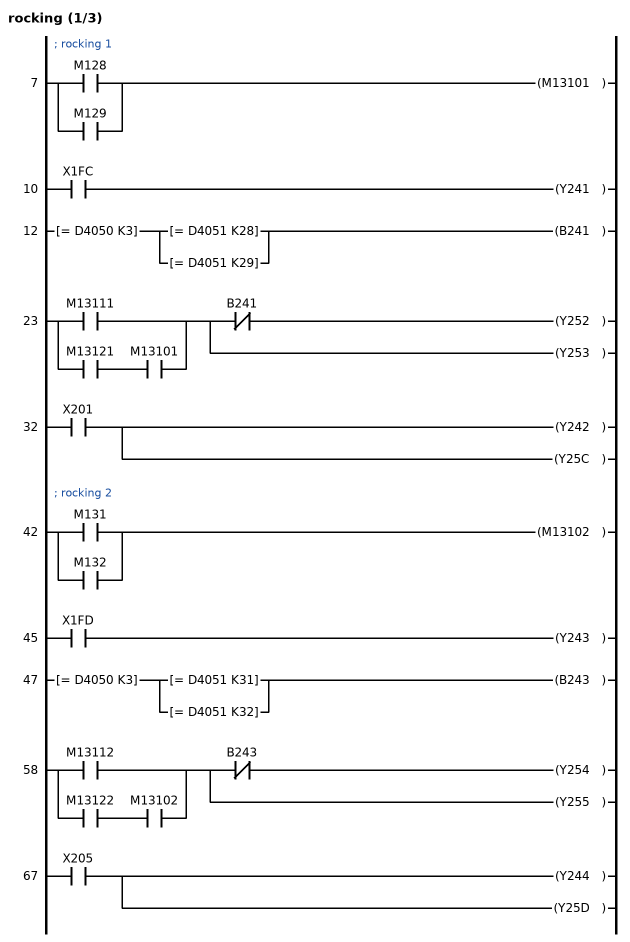
; rocking 1
7     LD      M128
      OR      M129
      OUT     M13101
10    LD      X1FC
      OUT     Y241
12    LD=     D4050 K3
      LD=     D4051 K28
      OR=     D4051 K29
      ANB
      OUT     B241
23    LD      M13111
      LD      M13121
      AND     M13101
      ORB
      MPS
      ANI     B241
      OUT     Y252
      MPP
      OUT     Y253
32    LD      X201
      OUT     Y242
      OUT     Y25C
; rocking 2
42    LD      M131
      OR      M132
      OUT     M13102
45    LD      X1FD
      OUT     Y243
47    LD=     D4050 K3
      LD=     D4051 K31
      OR=     D4051 K32
      ANB
      OUT     B243
58    LD      M13112
      LD      M13122
      AND     M13102
      ORB
      MPS
      ANI     B243
      OUT     Y254
      MPP
      OUT     Y255
67    LD      X205
      OUT     Y244
      OUT     Y25D
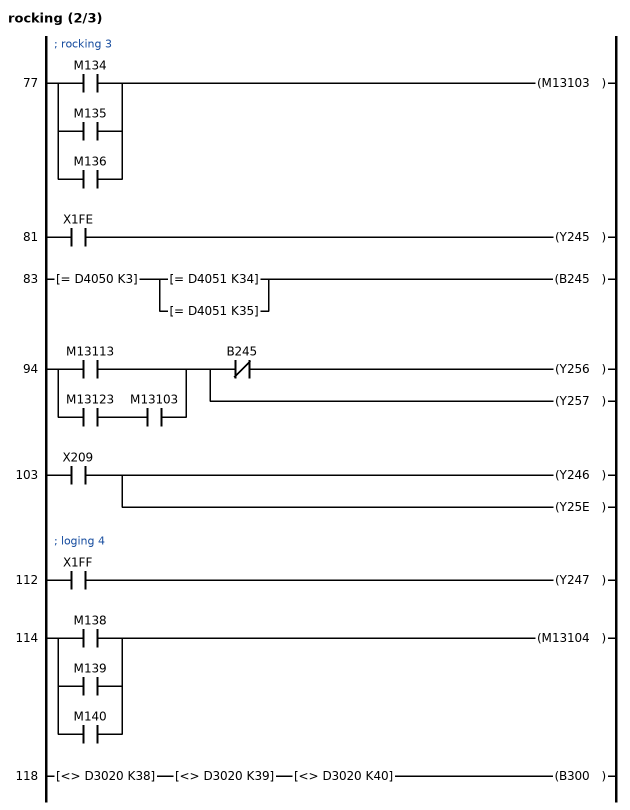
; rocking 3
77    LD      M134
      OR      M135
      OR      M136
      OUT     M13103
81    LD      X1FE
      OUT     Y245
83    LD=     D4050 K3
      LD=     D4051 K34
      OR=     D4051 K35
      ANB
      OUT     B245
94    LD      M13113
      LD      M13123
      AND     M13103
      ORB
      MPS
      ANI     B245
      OUT     Y256
      MPP
      OUT     Y257
103   LD      X209
      OUT     Y246
      OUT     Y25E
; loging 4
112   LD      X1FF
      OUT     Y247
114   LD      M138
      OR      M139
      OR      M140
      OUT     M13104
118   LD<>    D3020 K38
      AND<>   D3020 K39
      AND<>   D3020 K40
      OUT     B300
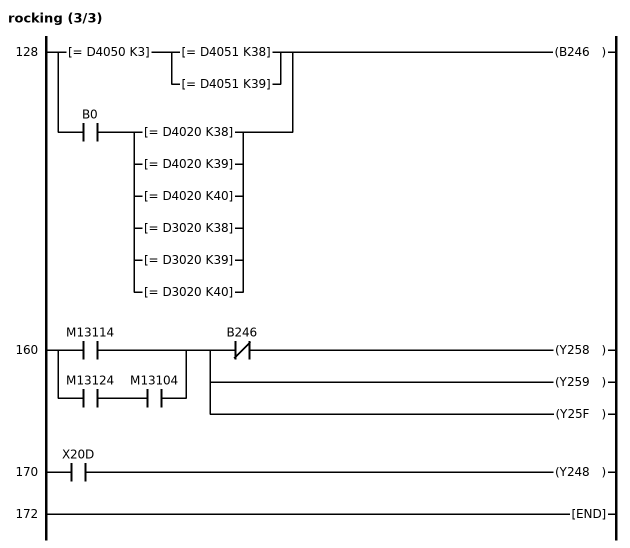
128   LD=     D4050 K3
      LD=     D4051 K38
      OR=     D4051 K39
      ANB
      LD      B0
      LD=     D4020 K38
      OR=     D4020 K39
      OR=     D4020 K40
      OR=     D3020 K38
      OR=     D3020 K39
      OR=     D3020 K40
      ANB
      ORB
      OUT     B246
160   LD      M13114
      LD      M13124
      AND     M13104
      ORB
      MPS
      ANI     B246
      OUT     Y258
      MPP
      OUT     Y259
      OUT     Y25F
170   LD      X20D
      OUT     Y248
172   END
END_PROGRAM

PROGRAM scrubber
